Staubli VAL3: Step1_Mount.pgx

program Step1_Mount()
  local bool l_bOut
  local num l_nKey
begin
  call ListMsg(true,"HMImount")
  l_bOut=false
  while !l_bOut
    do
      l_nKey=get()-270
    until l_nKey==1 or l_nKey==2 or l_nKey==7 or l_nKey==-15
    switch l_nKey
      case 1
        nMount=1
        sMount="floor"
        call ListMsg(true,"HMImount")
        call ListPop("Floor")
      break
      case 2
        nMount=-1
        sMount="ceiling"
        call ListMsg(true,"HMImount")
        call ListPop("Ceiling")
      break
      case 7,-15
        wait(getKey()==-1)
        call ListMsg(true,"HMImain")
        l_bOut=true
      break
    endSwitch
  endWhile
end
